TYPE ST_DigitalInputOutImm :
STRUCT
    Value : BOOL;
    Quality : BOOL;
    IoTag : STRING(80);
END_STRUCT
END_TYPE

(* stored: Version 1.1.0.1, ProductVersion 3.1.4024.12
   DUT ST_DigitalInputOutImm: Id {2a89f921-00cc-4be4-8027-e2c9b2ba3f95} *)
